RoboDK station: BendingCuadro.rdk

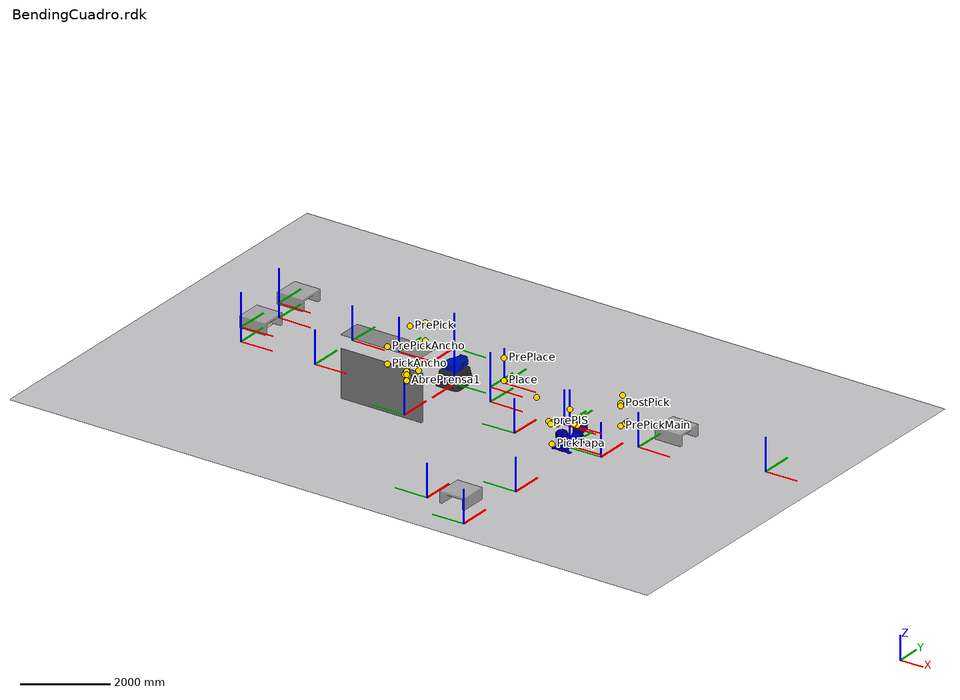
[picture v0: the station drawn from its stored meshes, robots at their saved joint values, targets as dots, program paths as lines]
Station BendingCuadro (saved by RoboDK 5.9.4). Poses are relative to the parent item; angles as X-Y-Z fixed-axis rotations.
Station parameters (name, value as stored): SensorCA, 0, SensorCL, 0, BendingHecho, 0, enCintaMain, 0, SensorCC, 0, EnMesa, 0, LasDos, 0
  - machining project Ajustes de mecanizado1: rotZ(0) | rotX(0)*rotY(0) | rotz(0) | onStart | onPathStart | onApproach | onPoint | onRetract | onFinish | SetRPM(%1) | SetTool(%1) | Extruder(%1) | default | default | OutOnMov(%1) | OutOffMov(%1) | onPathFinish | M_RunCode(%1)
  - folder Sistemas de Ref
    - frame World at (0, 0, 0) mm, rotated rx 0 ry 0 rz -90 deg
      - object Valla at (10, -2980, 0) mm, rotated rx 0 ry 0 rz 90 deg
      - object PedestalRobotPrensado at (0, 0, 0) mm, rotated rx 0 ry 0 rz 90 deg, size 633.4 x 700.2 x 375 mm, 1065353216 curves, geometry from Pedestal-H500mm-Type-2 (1).sld
      - object Suelo at (550, 1000, -5) mm, size 11520 x 17280 x 0 mm, 1056816382 curves, geometry from Suelo.stl
      - frame Frame_CintaCuadroInit at (300, 1190, 0) mm, rotated rx 0 ry 0 rz 90 deg
        - robot CintaCuadroIni: 1 axes
            modified DH rows (alpha deg, a mm, theta deg, d mm): 0, 0, 0, 0 linear
            base shift (0, 0, 0) mm, rotated rx 0 ry 90 rz 0 deg
            joint limits [-900000] to [900000]; home [0]; saved at [0]
          - frame FramePlanchaMain at (0, 0, 0) mm
      - frame Frame_CintaCuadroMid at (300, 3190, 0) mm, rotated rx 0 ry 0 rz 90 deg
        - robot CintaCuadroMid: 1 axes
            modified DH rows (alpha deg, a mm, theta deg, d mm): 0, 0, 0, 0 linear
            base shift (0, 0, 0) mm, rotated rx 0 ry 90 rz 0 deg
            joint limits [-900000] to [900000]; home [0]; saved at [0]
        - object SensorCC at (1240, 630, 370) mm, rotated rx 90 ry 0 rz -90 deg
      - frame Frame_CintaCuadroFinal at (300, 5190, 0) mm, rotated rx 0 ry 0 rz 90 deg
        - robot CintaCuadroFini: 1 axes
            modified DH rows (alpha deg, a mm, theta deg, d mm): 0, 0, 0, 0 linear
            base shift (0, 0, 0) mm, rotated rx 0 ry 90 rz 0 deg
            joint limits [-900000] to [900000]; home [0]; saved at [3450]
          - frame CuadroAcabada at (0, 0, 0) mm
        - target CintaCuadroSoldadoIni (joint target) at (-550, 0, 366.5) mm; joints [3450] of CintaCuadroFini
        - target CintaCuadroSoldadoFin (joint target) at (2010, 0, 366.5) mm; joints [6010, -103.845, 100.785, 0, -114.63, -14.149, 0] of CintaCuadroFini
        - object tunelCuadro at (-1600, 3110, 10) mm, size 688.9 x 676.6 x 291.3 mm, geometry from tunel.stl
      - frame Frame_CintaAnchoInit at (970, -5100, 0) mm, rotated rx 0 ry 0 rz 90 deg
        - robot CintaAnchoIni: 1 axes
            modified DH rows (alpha deg, a mm, theta deg, d mm): 0, 0, 0, 0 linear
            base shift (0, 0, 0) mm, rotated rx 0 ry 90 rz 0 deg
            joint limits [-900000] to [900000]; home [0]; saved at [0]
          - frame FramePlanchaAncha at (9, 0, 0) mm
            - object planxaAncha at (260, 305, 5) mm, size 467.5 x 467.7 x 2.1 mm, geometry from planxa1.2.stl
        - object tunelAcnha at (-2100, 3110, 10) mm, size 688.9 x 676.6 x 291.3 mm, geometry from tunel.stl
      - frame Frame_CintaAnchoFinal at (970, -3100, 0) mm, rotated rx 0 ry 0 rz 90 deg
        - robot Conveyor Belt Wide (2m): 1 axes
            modified DH rows (alpha deg, a mm, theta deg, d mm): 0, 0, 0, 0 linear
            base shift (0, 0, 0) mm, rotated rx 0 ry 90 rz 0 deg
            joint limits [-900000] to [900000]; home [0]; saved at [28.931]
        - object SensorCA at (1695, -40, 351.5) mm, rotated rx 90 ry 0 rz 90 deg
      - frame Frame_CintaLargoInit at (-490, -5100, 0) mm, rotated rx 0 ry 0 rz 90 deg
        - robot CintaLargoIni: 1 axes
            modified DH rows (alpha deg, a mm, theta deg, d mm): 0, 0, 0, 0 linear
            base shift (0, 0, 0) mm, rotated rx 0 ry 90 rz 0 deg
            joint limits [-900000] to [900000]; home [0]; saved at [0]
          - frame FramePlanchaLarga at (0, 0, 0) mm
            - object planxaLarga at (220, 310, 5) mm, size 294 x 630 x 2.1 mm, geometry from planxa1.3.stl
        - object tunelLarga at (-2100, 3110, 10) mm, size 688.9 x 676.6 x 291.3 mm, geometry from tunel.stl
      - frame Frame_CintaLargoFinal at (-490, -3100, 0) mm, rotated rx 0 ry 0 rz 90 deg
        - robot Conveyor Belt Wide (2m): 1 axes
            modified DH rows (alpha deg, a mm, theta deg, d mm): 0, 0, 0, 0 linear
            base shift (0, 0, 0) mm, rotated rx 0 ry 90 rz 0 deg
            joint limits [-900000] to [900000]; home [0]; saved at [28.931]
        - object SensorCL at (1645, -40, 351.5) mm, rotated rx 90 ry 0 rz 90 deg
      - frame Frame_CintaTapaInit at (5690, 4240, 0) mm, rotated rx 0 ry 0 rz 180 deg
        - robot CintaTapaInit: 1 axes
            modified DH rows (alpha deg, a mm, theta deg, d mm): 0, 0, 0, 0 linear
            base shift (0, 0, 0) mm, rotated rx 0 ry 90 rz 0 deg
            joint limits [-900000] to [900000]; home [0]; saved at [0]
          - frame FrameTapa at (0, 1000, 0) mm
        - object tunelTapa at (-2100, 3110, 10) mm, size 688.9 x 676.6 x 291.3 mm, geometry from tunel.stl
      - frame Frame_CintaTapaFinal at (3690, 4240, 0) mm, rotated rx 0 ry 0 rz 180 deg
        - robot CintaTapaFinal: 1 axes
            modified DH rows (alpha deg, a mm, theta deg, d mm): 0, 0, 0, 0 linear
            base shift (0, 0, 0) mm, rotated rx 0 ry 90 rz 0 deg
            joint limits [-900000] to [900000]; home [0]; saved at [3450]
        - object SensorTapa at (1550, 0, 370) mm, rotated rx 90 ry 0 rz 90 deg
    - frame RobotPrensado at (0, 0, 880) mm, rotated rx 0 ry 0 rz -90 deg
      - robot Yaskawa MH24 Prensado (model Yaskawa MH24): 6 axes, payload 24 kg, reach 1730 mm, repeatability 0.06 mm, weight 268 kg
          modified DH rows (alpha deg, a mm, theta deg, d mm): 0, 0, 0, 505; -90, 150, -90, 0; 0, 760, 0, 0; -90, 200, 0, 795; 90, 0, 0, 0; -90, 0, 0, 100
          base shift (0, 0, -505) mm
          joint limits [-180, -105, -170, -200, -150, -455] to [180, 155, 240, 200, 150, 455]; home [0, 0, 0, 0, 0, 0]; saved at [0, 39.675, 3.651, 0, -56.577, 90]
        - tool EPick Bend, TCP at (0, 0, 185) mm
    - frame RobotPaletizado at (4800, -1180, 0) mm, rotated rx 0 ry 0 rz 90 deg
      - robot ABB Paletizado (model ABB IRB 1660-4/1.55): 6 axes, payload 4 kg, reach 1550 mm, repeatability 0.02 mm, weight 257 kg
          modified DH rows (alpha deg, a mm, theta deg, d mm): 0, 0, 0, 481.5; -90, 150, -90, 0; 0, 700, 0, 0; -90, 110, 0, 678; 90, 0, 0, 0; -90, 0, 180, 135
          joint limits [-180, -90, -238, -175, -120, -400] to [180, 150, 79, 175, 120, 400]; home [0, 0, 0, 0, 0, 0]; saved at [0, -27.309, 31.419, 0, -4.109, 90]
        - tool EPick Gripper, TCP at (0, 30, 180) mm
      - frame Cinta_Mesa at (0, 0, 0) mm
        - target PrePickMain (Cartesian target) at (768.94, -0.74, 460.56) mm, rotated rx 88.94 ry 0.2 rz 90.33 deg; joints [-0.34, 25.821, 73.422, -0.689, -100.301, 89.691, 0] of ABB Paletizado
        - target PickMainLarga (Cartesian target) at (933.91, 0.24, 463.61) mm, rotated rx 88.94 ry 0.2 rz 90.33 deg; joints [-0.159, 27.939, 59.383, -0.497, -88.381, 89.825, 0] of ABB Paletizado
        - target PickMainAncha (Cartesian target) at (1018.89, 0.74, 465.18) mm, rotated rx 88.94 ry 0.2 rz 90.33 deg; joints [-0.099, 30.281, 51.872, -0.44, -83.211, 89.862, 0] of ABB Paletizado
        - target PostPick (Cartesian target) at (758.49, 1.16, 1025.46) mm, rotated rx 88.94 ry 0.2 rz 90.33 deg; joints [-0.104, -33.737, 49.135, -1.559, -16.462, 91.305, 0] of ABB Paletizado
        - target Giro180_P (Cartesian target) at (759.67, 0.31, 965.48) mm, rotated rx -88.95 ry -1.49 rz -89.69 deg; joints [-0.1, -33.73, 49.13, -1.55, -16.46, -90, 0] of ABB Paletizado
        - target PrePlaceMain (Cartesian target) at (34.68, 675.75, 588.97) mm, rotated rx -88.96 ry -1.48 rz -1.79 deg; joints [86.158, -18.643, 78.562, -2.38, -60.986, -90.292, 0] of ABB Paletizado
        - target PlaceMain (Cartesian target) at (36.98, 750.71, 590.34) mm, rotated rx -88.96 ry -1.48 rz -1.79 deg; joints [86.516, -9.473, 72.928, -1.909, -64.513, -90.631, 0] of ABB Paletizado
      - target Inicio (Cartesian target) at (827.98, 0, 1194.61) mm, rotated rx 90 ry 0 rz 90 deg; joints [0, -27.309, 31.419, 0, -4.109, 90, 0] of ABB Paletizado
      - target PrePickCuadro (Cartesian target) at (4.9, 841.7, 940.96) mm, rotated rx 179.08 ry 0.41 rz 174.95 deg; joints [90.03, -2.117, 5.113, -0.49, 86.121, 95.109, 0] of ABB Paletizado
      - target PickCuadro (Cartesian target) at (4.9, 841.7, 680.96) mm, rotated rx 179.08 ry 0.41 rz 174.95 deg; joints [90.03, -0.345, 25.277, -0.543, 64.186, 95.312, 0] of ABB Paletizado
      - target PrePickTapa (Cartesian target) at (-778.15, 778.56, 940.96) mm, rotated rx -179.33 ry -0.3 rz -86.95 deg; joints [133.893, 21.723, -22.95, -0.311, 91.887, 40.834, 0] of ABB Paletizado
      - target PickTapa (Cartesian target) at (-778.15, 778.56, 412.42) mm, rotated rx -179.33 ry -0.3 rz -86.95 deg; joints [133.893, 29.971, 10.868, -0.407, 49.822, 41.107, 0] of ABB Paletizado
    - frame RobotSoldador at (2530, -1300, 0) mm, rotated rx 0 ry 0 rz 90 deg
      - robot ABB Soldador (model ABB IRB 1660-4/1.55): 6 axes, payload 4 kg, reach 1550 mm, repeatability 0.02 mm, weight 257 kg
          modified DH rows (alpha deg, a mm, theta deg, d mm): 0, 0, 0, 481.5; -90, 150, -90, 0; 0, 700, 0, 0; -90, 110, 0, 678; 90, 0, 0, 0; -90, 0, 180, 135
          joint limits [-180, -90, -238, -175, -120, -400] to [180, 150, 79, 175, 120, 400]; home [0, 0, 0, 0, 0, 0]; saved at [180, 5.81, -214.75, 0, 0, 0]
        - tool Welding Gun, TCP at (86, 0, 451.5) mm, rotated rx 0 ry 36 rz 0 deg
      - target Inicio_Soldador (Cartesian target) at (874.12, 0, 545.02) mm, rotated rx 0 ry -82.94 rz 180 deg; joints [180, 5.81, -214.75, 0, 0, 0, 0] of ABB Soldador
      - target prePIS (Cartesian target) at (-101.3, -1007.69, 623.69) mm, rotated rx 134.47 ry 88.84 rz 90.8 deg; joints [53.05, -51.812, -173.339, -59.361, 109.58, -131.05, 0] of ABB Soldador
      - target PIS (Cartesian target) at (36.12, -1138.87, 621.01) mm, rotated rx 134.47 ry 88.84 rz 90.8 deg; joints [65.969, -54.136, -168.246, -51.218, 100.348, -134.197, 0] of ABB Soldador
      - target PFS (Cartesian target) at (36.09, -1137.26, 541.02) mm, rotated rx 134.47 ry 88.84 rz 90.8 deg; joints [65.922, -59.336, -166.814, -51.849, 102.718, -137.187, 0] of ABB Soldador
      - target postPFS (Cartesian target) at (-72.39, -1033.69, 543.14) mm, rotated rx 134.47 ry 88.84 rz 90.8 deg; joints [55.809, -57.49, -171.254, -58.794, 109.811, -135.353, 0] of ABB Soldador
    - frame Pick at (-1500, 0, 370) mm
      - target PrePick (Cartesian target) at (160, 190, 600) mm, rotated rx -180 ry 0 rz -90 deg; joints [-98.253, 31.893, -1.848, 0, -56.259, 98.253, 0] of Yaskawa MH24 Prensado
      - target PrePickAncho (Cartesian target) at (160, -670, 440) mm, rotated rx -180 ry 0 rz -90 deg; joints [-63.435, 49.441, 15.409, 180, 55.968, -116.565, 0] of Yaskawa MH24 Prensado
      - target PrePickLargo (Cartesian target) at (160, 790, 440) mm, rotated rx -180 ry 0 rz -90 deg; joints [-120.522, 54.399, 24.171, 0, -59.772, 120.522, 0] of Yaskawa MH24 Prensado
      - target PickAncho (Cartesian target) at (160, -670, 0) mm, rotated rx -180 ry 0 rz -90 deg; joints [-63.435, 68.099, 15.642, 180, 37.543, -116.565, 0] of Yaskawa MH24 Prensado
      - target PickLargo (Cartesian target) at (160, 790, 0) mm, rotated rx -180 ry 0 rz -90 deg; joints [-120.522, 72.326, 24.429, 180, 42.104, -59.478, 0] of Yaskawa MH24 Prensado
    - frame Place at (1350, 0, 400) mm
      - target PrePlace (Cartesian target) at (0, 0, 610) mm, rotated rx -180 ry 0 rz 90 deg; joints [90, 30.642, -0.787, 0, -58.571, 90, 0] of Yaskawa MH24 Prensado
      - target Place (Cartesian target) at (0, 0, 56) mm, rotated rx 180 ry 0 rz 90 deg; joints [90, 53.307, -7.669, -180, 29.024, 270, 0] of Yaskawa MH24 Prensado
    - frame MesaGiratoria at (3900, -1100, 0) mm
      - robot Yaskawa Giratoria (model Motoman MOTOPOS-D250F): 2 axes
          modified DH rows (alpha deg, a mm, theta deg, d mm): 0, 0, 0, 0; 90, 0, 0, 0
          base shift (0, 0, 380) mm, rotated rx -90 ry 0 rz 0 deg
          joint limits [-135, -200] to [135, 200]; home [0, 0]; saved at [0, 0]
        - frame Engranaje at (0, 0, 0) mm
          - object planchaAcabada at (-360, 520, 370) mm, rotated rx 0 ry 0 rz 90 deg, size 297.8 x 466.8 x 85.5 mm, geometry from planchaAcabada.stl
      - target Inici (Cartesian target) at (0, 0, 530) mm; joints [0, 0, -7.748, -180, 29.277, 270, 0] of Yaskawa Giratoria
      - target Giro90 (joint target) at (0, 0, 530) mm, rotated rx 0 ry 0 rz 90 deg; joints [0, 90, 19.031, 0, -41.803, 121.092, 0] of Yaskawa Giratoria
      - target Esquina0 (Cartesian target) at (0, 0, 530) mm, rotated rx 0 ry 0 rz -90 deg; joints [0, -90, 0, 0, 0, 0, 0] of Yaskawa Giratoria
      - target Esquina1 (Cartesian target) at (0, 0, 530) mm, rotated rx 0 ry 0 rz -22.95 deg; joints [0, -22.95, 0, 0, 0, 0, 0] of Yaskawa Giratoria
      - target Esquina2 (Cartesian target) at (0, 0, 530) mm, rotated rx 0 ry 0 rz 90 deg; joints [0, 90, 0, 0, 0, 0, 0] of Yaskawa Giratoria
      - target Esquina3 (Cartesian target) at (0, 0, 530) mm, rotated rx 0 ry 0 rz 157.38 deg; joints [0, 157.38, 0, 0, 0, 0, 0] of Yaskawa Giratoria
      - target Final (Cartesian target) at (0, 0, 530) mm, rotated rx 0 ry 0 rz 180 deg; joints [0, 180, -7.748, -180, 29.277, 270, 0] of Yaskawa Giratoria
    - frame Bending at (0, -1940, 0) mm, rotated rx 0 ry 0 rz 90 deg
      - object tapa_prensa at (-450, 120, 1965) mm, size 640 x 2140 x 5 mm, geometry from tapa_prensa3.stl
      - object tapa_darrere at (-725, 110, 990) mm, rotated rx 0 ry 0 rz 90 deg, size 2197.8 x 29.7 x 1217.7 mm, 1064168942 curves, geometry from tapaor3.stl
      - robot Press Brake: 1 axes
          modified DH rows (alpha deg, a mm, theta deg, d mm): 0, 0, 0, 0 linear
          joint limits [0] to [230]; home [0]; saved at [0]
      - target Home (Cartesian target) at (557.12, 0, 874.46) mm, rotated rx -177.4 ry 0 rz -90 deg; joints [0, 37.6, 0, 0, -55, 90, 0] of Yaskawa MH24 Prensado
      - target Place1 (joint target) at (144.16, 0, 929.49) mm, rotated rx 0 ry -31.66 rz 0 deg; joints [0, 79.41, 41.34, 0, 96.41, 0, 0] of Yaskawa MH24 Prensado
      - target Place2 (joint target) at (144.16, 0, 929.49) mm, rotated rx 0 ry 31.66 rz -180 deg; joints [0, 79.41, 41.34, 0, 96.41, 180, 0] of Yaskawa MH24 Prensado
      - target BajaPrensa1 (joint target) at (144.16, 0, 929.49) mm, rotated rx 0 ry -31.66 rz 0 deg; joints [0, 79.41, 41.34, 0, 96.41, 0, 230] of Yaskawa MH24 Prensado
      - target BajaPrensa2 (joint target) at (144.16, 0, 1159.49) mm, rotated rx 0 ry 31.66 rz -180 deg; joints [0, 79.41, 41.34, 0, 96.41, 180, 230] of Yaskawa MH24 Prensado
      - target Bend1 (joint target) at (101.51, 0, 1035) mm, rotated rx 0 ry -60 rz 0 deg; joints [0, 64.383, 27.581, 0, 66.801, 0, 230] of Yaskawa MH24 Prensado
      - target BendA1 (joint target) at (57.18, 30, 968.22) mm, rotated rx 0 ry -60 rz 0 deg; joints [0, 71.944, 37.304, 0, 64.64, 0, 230] of Yaskawa MH24 Prensado
      - target Bend2 (joint target) at (101.52, 0, 1035.05) mm, rotated rx 0 ry 60 rz -180 deg; joints [0, 64.38, 27.58, 0, 66.8, 180, 230] of Yaskawa MH24 Prensado
      - target BendA2 (joint target) at (65.36, -30, 970.72) mm, rotated rx 0 ry 60 rz -180 deg; joints [0, 70.932, 35.526, 0, 65.405, 180, 230] of Yaskawa MH24 Prensado
      - target AbrePrensa1 (joint target) at (101.51, 0, 805) mm, rotated rx 0 ry -60.01 rz 0 deg; joints [0, 64.378, 27.576, 0, 66.792, 0, 0] of Yaskawa MH24 Prensado
      - target AbrePrensa2 (joint target) at (101.49, 0, 805) mm, rotated rx 0 ry 60.01 rz -180 deg; joints [0, 64.38, 27.58, 0, 66.79, 180, 0] of Yaskawa MH24 Prensado
      - target Retract1 (Cartesian target) at (485.32, 30, 1066.8) mm, rotated rx -180 ry -87.45 rz 180 deg; joints [0, 27.86, -21.47, 0, 46.78, 0, 0] of Yaskawa MH24 Prensado
      - target Retract2 (Cartesian target) at (488.99, -30, 1096.85) mm, rotated rx -180 ry 87.44 rz 0 deg; joints [0, 26.34, -21.22, 0, 45, -180, 0] of Yaskawa MH24 Prensado
      - target Gir180 (Cartesian target) at (482.67, -30, 1126.45) mm, rotated rx 180 ry 87.43 rz 0 deg; joints [0, 25.54, -19.95, 0, 42.92, 180, 0] of Yaskawa MH24 Prensado
      - object planchaAncha1 at (51.51, 30, 965) mm, rotated rx 0 ry 60 rz 180 deg, size 379 x 462.2 x 85.1 mm, geometry from planxa2.3._intermig.stl
      - object planchaLarga1 at (101.51, 30, 1035) mm, rotated rx -60 ry 0 rz 90 deg, size 294 x 547 x 85.1 mm, geometry from planxa2.2_intermig.stl
      - object planchaLarga2 at (100.51, -30, 1035) mm, rotated rx -60 ry 0 rz 90 deg, size 294 x 464.1 x 85.1 mm, geometry from planxa2.2.stl
      - object planchaAncha2 at (51.51, -30, 965) mm, rotated rx 0 ry 60 rz 180 deg, size 296.1 x 462.2 x 85.1 mm, geometry from planxa2.1.stl
  - folder Programas
    - program RESET (7 instructions, listed below)
    - Python program main (listed below)
    - Python program reset (listed below)

--- program RESET ---
  Reemplazar planxaLarga
  Reemplazar planchaLarga1
  Reemplazar planchaLarga2
  Reemplazar planxaAncha
  Reemplazar planchaAncha1
  Reemplazar planchaAncha2
  Reemplazar planchaAcabada

--- Python program main ---
import threading
import traceback
from modulos_python.entorno import preparar_entorno

preparar_entorno()

from modulos_python import pick, place, bending, soldar, sensor, var
from modulos_python import mover_cintas as mc
from robodk import robolink
from robodk import robomath

def getIniPose():
    RDK = robolink.Robolink()
    lista_ini_objetos = RDK.ItemList(robolink.ITEM_TYPE_OBJECT)

    for idx in lista_ini_objetos:
        if isinstance(idx, str):
            idx = RDK.Item(idx)

        var.registrar_info_objeto_json(idx.Name(), str(idx.Pose()), str(idx.Parent()))

getIniPose()
robomath.pause(1)

def _thread_excepthook(args):
    RDK = robolink.Robolink()

    RDK.ShowMessage(f"[ThreadError] {args.thread.name}: {args.exc_type.__name__}: {args.exc_value}")
    traceback.print_exception(args.exc_type, args.exc_value, args.exc_traceback)

threading.excepthook = _thread_excepthook

def hilo_cinta_larga():
    mc.mover_cinta_larga()

def hilo_cinta_ancha():
    mc.mover_cinta_ancha()

def hilo_cinta_tapa():
    mc.mover_cinta_tapa()

def hilo_yaskawa():
    """ que piezas pendientes tengo en cola """

    RDK = robolink.Robolink()

    ultima = None

    cola_ancha = var.objetos_pendientes["SensorCA"]
    cola_larga = var.objetos_pendientes["SensorCL"]

    while True:

        if ultima is None:
            if not cola_ancha.empty():
                obj1 = cola_ancha.get()
                pick.pick_plancha_ancha()

                if obj1 is not None:
                    RDK.ShowMessage(f"objeto consumido: {obj1.Name()}", False)

                bending.bending_plancha_ancha()
                place.place_cinta_main()
                ultima = "ancha"
                var.alternancia.put(ultima)

            elif not cola_larga.empty():
                obj2 = cola_larga.get()
                pick.pick_plancha_larga()

                if obj2 is not None:
                    RDK.ShowMessage(f"objeto consumido: {obj2.Name()}", False)

                bending.bending_plancha_larga()
                place.place_cinta_main()
                ultima = "larga"
                var.alternancia.put(ultima)
            else:
                RDK.ShowMessage(f"no esta haciendo nada el hilo_yaskawa", False)
                robomath.pause(0.01)
        elif ultima == "ancha":
                if not cola_larga.empty():
                    obj2 = cola_larga.get()
                    pick.pick_plancha_larga()

                    if obj2 is not None:
                        RDK.ShowMessage(f"objeto consumido: {obj2.Name()}", False)

                    bending.bending_plancha_larga()
                    place.place_cinta_main()
                    ultima = "larga"
                    var.alternancia.put(ultima)
        elif ultima == "larga":
                if not cola_ancha.empty():
                    obj1 = cola_ancha.get()
                    pick.pick_plancha_ancha()

                    if obj1 is not None:
                        RDK.ShowMessage(f"objeto consumido: {obj1.Name()}", False)

                    bending.bending_plancha_ancha()
                    place.place_cinta_main()
                    ultima = "ancha"
                    var.alternancia.put(ultima)
        else:
            robomath.pause(0.01)


def hilo_cinta_main():
    RDK = robolink.Robolink()
    while True:
        mc.mover_cinta_main(RDK)

def hilo_place_mesa():
    while True:
        place.place_plancha_mesa()

def hilo_place_soldado():
    while True:
        place.place_plancha_soldada()

def hilo_soldador():
    while True:
        soldar.soldar_ini()

def hilo_sensorCA():
    sensor.detectar_objeto("SensorCA", "FramePlanchaAncha")

def hilo_sensorCL():
    sensor.detectar_objeto("SensorCL", "FramePlanchaLarga")

def hilo_sensorCC():
    sensor.detectar_objeto("SensorCC", "FramePlanchaMain")

def hilo_sensorTapa():
    sensor.detectar_objeto("SensorTapa", "FrameTapa")

threads = [
    threading.Thread(target=hilo_cinta_larga, name="cinta_larga"),
    threading.Thread(target=hilo_cinta_ancha, name="cinta_ancha"),
    threading.Thread(target=hilo_cinta_tapa, name="cinta_tapa"),
    threading.Thread(target=hilo_yaskawa, name="yaskawa"),
    threading.Thread(target=hilo_cinta_main, name="cinta_main"),
    threading.Thread(target=hilo_place_mesa, name="place_mesa"),
    threading.Thread(target=hilo_place_soldado, name="place_soldado"),
    threading.Thread(target=hilo_soldador, name="soldador"),
    threading.Thread(target=hilo_sensorCA, name="sensor_ca"),
    threading.Thread(target=hilo_sensorCL, name="sensor_cl"),
    threading.Thread(target=hilo_sensorCC, name="sensor_cc"),
    threading.Thread(target=hilo_sensorTapa, name="sensor_tapa")
]

for t in threads:
    t.start()

--- Python program reset ---
from robodk import robolink
from robodk import robomath
from modulos_python import simulation, var
import json

def reset_cinta(nombre_cinta : str):
    RDK = robolink.Robolink()

    item_cinta = RDK.Item(nombre_cinta, robolink.ITEM_TYPE_ROBOT)
    if not item_cinta.Valid():
        raise RuntimeError(RDK.ShowMessage(f"Cinta: {nombre_cinta} no existe, revisa nombres"))

    item_cinta.setJoints(robomath.Mat([[0]]))

def reset_param():
    if not var.JSON_PARAM_PATH.exists():
        return
    with var.JSON_PARAM_PATH.open("r", encoding="utf-8") as f:
        data = json.load(f)

    parametros = data.get("parametros", []) if isinstance(data, dict) else data
    for nombre in parametros:
        simulation.setDO(str(nombre), 0)

def reset_objetos():
    if not var.JSON_PARAM_PATH.exists():
        return
    with var.JSON_PARAM_PATH.open("r", encoding="utf-8") as f:
        data = json.load(f)

    info_objetos = data.get("info_objetos", {}) if isinstance(data, dict) else data
    for nombre in info_objetos:
        simulation.reemplazar_pos_objeto(nombre[0], nombre[1], nombre[2])

reset_param()
#reset_objetos()

reset_cinta(var.cinta_larga)
reset_cinta(var.cinta_ancha)
reset_cinta(var.cinta_main)
reset_cinta(var.cinta_tapa)
reset_cinta(var.mesa_giratoria)

simulation.mostrar_objeto("planxaLarga")
simulation.mostrar_objeto("planxaAncha")

simulation.ocultar_objeto("planchaLarga2")
simulation.ocultar_objeto("planchaAncha2")
simulation.ocultar_objeto("planchaAcabada")
